// TIA Portal V17 export
// export: Created 2025-03-07T09:17:15.516667Z, ExportSetting WithDefaults, DisplayName Totally Integrated Automation Portal, DisplayVersion V17 Update 8, DisplayName TIA Portal Openness, DisplayVersion V17 Update 8, DisplayName TIA Portal Version Control Interface, DisplayVersion V17, DisplayName SINAMICS Startdrive Advanced, DisplayVersion V17 SP2, DisplayName SINAMICS Startdrive G110M, G120, G120C, G120D, G120P, G115D, DisplayVersion V17 SP2, DisplayName SINAMICS Startdrive G130, G150, S120, S150, SINAMICS MV, S210, DisplayVersion V17 SP2, DisplayName STEP 7 Professional, DisplayVersion V17 Update 8, DisplayName SINUMERIK ONE STEP 7 Toolbox, DisplayVersion V17 Update 12, DisplayName SINUMERIK 840D sl STEP 7 Toolbox, DisplayVersion V17 Update 12, DisplayName STEP 7 Safety, DisplayVersion V17 Update 6, DisplayName WinCC Advanced, DisplayVersion V17 Update 8
FUNCTION "FC355_NCK_M_CH3_UNIT_1_STA_4" : Void   // FC355, LAD
TITLE = Channel 1 data
{ S7_Optimized_Access := 'FALSE' }
AUTHOR : ETXETAR
VERSION : 1.0
// stored: AutoNumber false, IsIECCheckEnabled false, SetENOAutomatically false, UDAEnableTagReadback false
BEGIN

REGION Network 1: ACKNOWLEDGE M700-FIXTURE 4 CLAMP SEQUENCE (READ-IN DISABLE) / ACKNOWLEDGE M100-CLAMP SEQUENCE FIXTURE 1
   // NOTE: WHEN THERE IS NOT INDEXING TABLE AVAILABLE IN THE MACHINE DELETE 
   // DB2171.DBX5.0 AND DB2171.DBX2.0
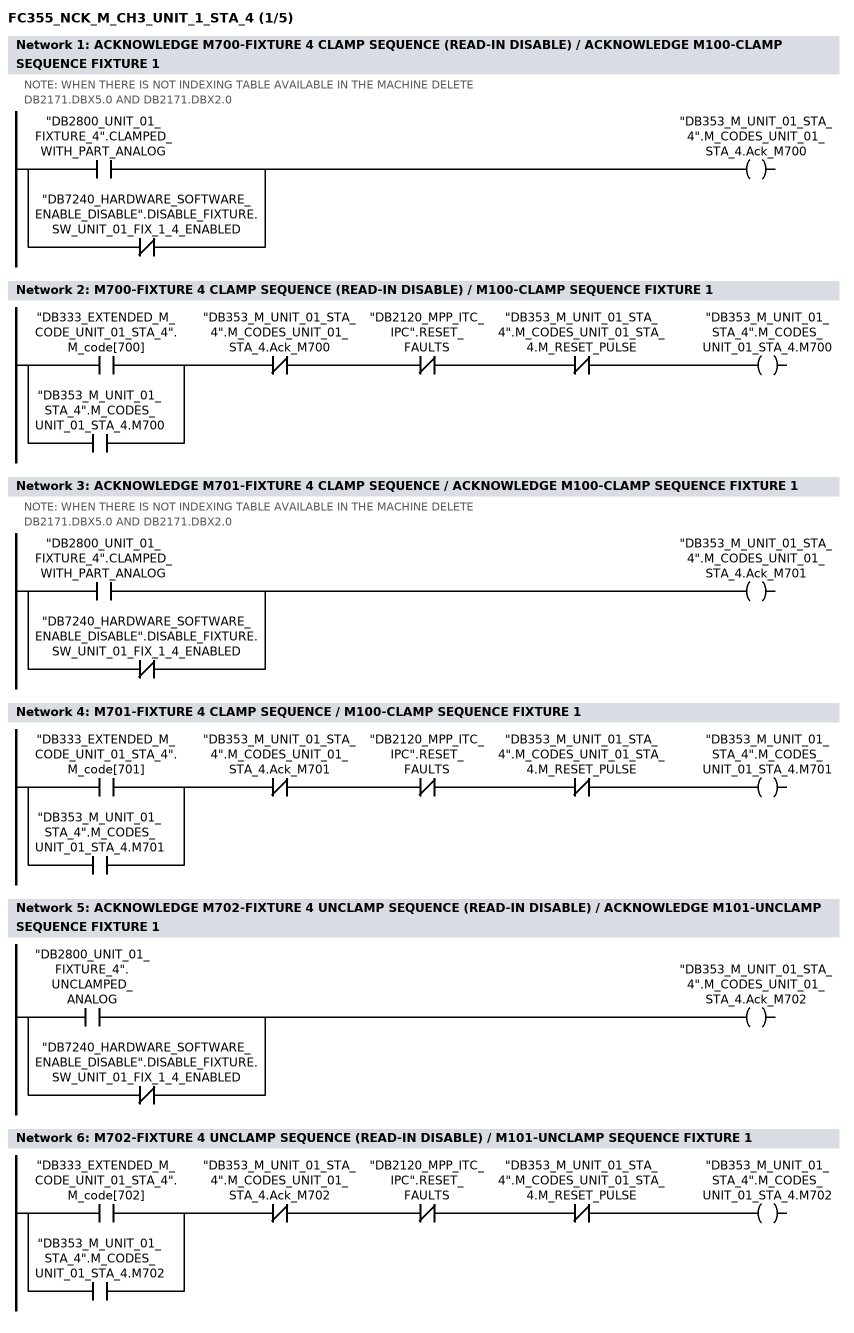
   RUNG wire#powerrail
      Contact( "DB2800_UNIT_01_FIXTURE_4".CLAMPED_WITH_PART_ANALOG )
      wire#w1
      Coil( "DB353_M_UNIT_01_STA_4".M_CODES_UNIT_01_STA_4.Ack_M700 )
   END_RUNG
   RUNG wire#powerrail
      I_Contact( "DB7240_HARDWARE_SOFTWARE_ENABLE_DISABLE".DISABLE_FIXTURE.SW_UNIT_01_FIX_1_4_ENABLED )
   END_RUNG wire#w1
   // the same network as SCL:
   "DB353_M_UNIT_01_STA_4".M_CODES_UNIT_01_STA_4.Ack_M700 := "DB2800_UNIT_01_FIXTURE_4".CLAMPED_WITH_PART_ANALOG OR NOT "DB7240_HARDWARE_SOFTWARE_ENABLE_DISABLE".DISABLE_FIXTURE.SW_UNIT_01_FIX_1_4_ENABLED;
END_REGION

REGION Network 2: M700-FIXTURE 4 CLAMP SEQUENCE (READ-IN DISABLE) / M100-CLAMP SEQUENCE FIXTURE 1
   RUNG wire#powerrail
      Contact( "DB333_EXTENDED_M_CODE_UNIT_01_STA_4".M_code[700] )
      wire#w1
      I_Contact( "DB353_M_UNIT_01_STA_4".M_CODES_UNIT_01_STA_4.Ack_M700 )
      I_Contact( "DB2120_MPP_ITC_IPC".RESET_FAULTS )
      I_Contact( "DB353_M_UNIT_01_STA_4".M_CODES_UNIT_01_STA_4.M_RESET_PULSE )
      Coil( "DB353_M_UNIT_01_STA_4".M_CODES_UNIT_01_STA_4.M700 )
   END_RUNG
   RUNG wire#powerrail
      Contact( "DB353_M_UNIT_01_STA_4".M_CODES_UNIT_01_STA_4.M700 )
   END_RUNG wire#w1
   // the same network as SCL:
   "DB353_M_UNIT_01_STA_4".M_CODES_UNIT_01_STA_4.M700 := ("DB333_EXTENDED_M_CODE_UNIT_01_STA_4".M_code[700] OR "DB353_M_UNIT_01_STA_4".M_CODES_UNIT_01_STA_4.M700) AND NOT "DB353_M_UNIT_01_STA_4".M_CODES_UNIT_01_STA_4.Ack_M700 AND NOT "DB2120_MPP_ITC_IPC".RESET_FAULTS AND NOT "DB353_M_UNIT_01_STA_4".M_CODES_UNIT_01_STA_4.M_RESET_PULSE;
END_REGION

REGION Network 3: ACKNOWLEDGE M701-FIXTURE 4 CLAMP SEQUENCE / ACKNOWLEDGE M100-CLAMP SEQUENCE FIXTURE 1
   // NOTE: WHEN THERE IS NOT INDEXING TABLE AVAILABLE IN THE MACHINE DELETE 
   // DB2171.DBX5.0 AND DB2171.DBX2.0
   RUNG wire#powerrail
      Contact( "DB2800_UNIT_01_FIXTURE_4".CLAMPED_WITH_PART_ANALOG )
      wire#w1
      Coil( "DB353_M_UNIT_01_STA_4".M_CODES_UNIT_01_STA_4.Ack_M701 )
   END_RUNG
   RUNG wire#powerrail
      I_Contact( "DB7240_HARDWARE_SOFTWARE_ENABLE_DISABLE".DISABLE_FIXTURE.SW_UNIT_01_FIX_1_4_ENABLED )
   END_RUNG wire#w1
   // the same network as SCL:
   "DB353_M_UNIT_01_STA_4".M_CODES_UNIT_01_STA_4.Ack_M701 := "DB2800_UNIT_01_FIXTURE_4".CLAMPED_WITH_PART_ANALOG OR NOT "DB7240_HARDWARE_SOFTWARE_ENABLE_DISABLE".DISABLE_FIXTURE.SW_UNIT_01_FIX_1_4_ENABLED;
END_REGION

REGION Network 4: M701-FIXTURE 4 CLAMP SEQUENCE / M100-CLAMP SEQUENCE FIXTURE 1
   RUNG wire#powerrail
      Contact( "DB333_EXTENDED_M_CODE_UNIT_01_STA_4".M_code[701] )
      wire#w1
      I_Contact( "DB353_M_UNIT_01_STA_4".M_CODES_UNIT_01_STA_4.Ack_M701 )
      I_Contact( "DB2120_MPP_ITC_IPC".RESET_FAULTS )
      I_Contact( "DB353_M_UNIT_01_STA_4".M_CODES_UNIT_01_STA_4.M_RESET_PULSE )
      Coil( "DB353_M_UNIT_01_STA_4".M_CODES_UNIT_01_STA_4.M701 )
   END_RUNG
   RUNG wire#powerrail
      Contact( "DB353_M_UNIT_01_STA_4".M_CODES_UNIT_01_STA_4.M701 )
   END_RUNG wire#w1
   // the same network as SCL:
   "DB353_M_UNIT_01_STA_4".M_CODES_UNIT_01_STA_4.M701 := ("DB333_EXTENDED_M_CODE_UNIT_01_STA_4".M_code[701] OR "DB353_M_UNIT_01_STA_4".M_CODES_UNIT_01_STA_4.M701) AND NOT "DB353_M_UNIT_01_STA_4".M_CODES_UNIT_01_STA_4.Ack_M701 AND NOT "DB2120_MPP_ITC_IPC".RESET_FAULTS AND NOT "DB353_M_UNIT_01_STA_4".M_CODES_UNIT_01_STA_4.M_RESET_PULSE;
END_REGION

REGION Network 5: ACKNOWLEDGE M702-FIXTURE 4 UNCLAMP SEQUENCE (READ-IN DISABLE) / ACKNOWLEDGE M101-UNCLAMP SEQUENCE FIXTURE 1
   RUNG wire#powerrail
      Contact( "DB2800_UNIT_01_FIXTURE_4".UNCLAMPED_ANALOG )
      wire#w1
      Coil( "DB353_M_UNIT_01_STA_4".M_CODES_UNIT_01_STA_4.Ack_M702 )
   END_RUNG
   RUNG wire#powerrail
      I_Contact( "DB7240_HARDWARE_SOFTWARE_ENABLE_DISABLE".DISABLE_FIXTURE.SW_UNIT_01_FIX_1_4_ENABLED )
   END_RUNG wire#w1
   // the same network as SCL:
   "DB353_M_UNIT_01_STA_4".M_CODES_UNIT_01_STA_4.Ack_M702 := "DB2800_UNIT_01_FIXTURE_4".UNCLAMPED_ANALOG OR NOT "DB7240_HARDWARE_SOFTWARE_ENABLE_DISABLE".DISABLE_FIXTURE.SW_UNIT_01_FIX_1_4_ENABLED;
END_REGION

REGION Network 6: M702-FIXTURE 4 UNCLAMP SEQUENCE (READ-IN DISABLE) / M101-UNCLAMP SEQUENCE FIXTURE 1
   RUNG wire#powerrail
      Contact( "DB333_EXTENDED_M_CODE_UNIT_01_STA_4".M_code[702] )
      wire#w1
      I_Contact( "DB353_M_UNIT_01_STA_4".M_CODES_UNIT_01_STA_4.Ack_M702 )
      I_Contact( "DB2120_MPP_ITC_IPC".RESET_FAULTS )
      I_Contact( "DB353_M_UNIT_01_STA_4".M_CODES_UNIT_01_STA_4.M_RESET_PULSE )
      Coil( "DB353_M_UNIT_01_STA_4".M_CODES_UNIT_01_STA_4.M702 )
   END_RUNG
   RUNG wire#powerrail
      Contact( "DB353_M_UNIT_01_STA_4".M_CODES_UNIT_01_STA_4.M702 )
   END_RUNG wire#w1
   // the same network as SCL:
   "DB353_M_UNIT_01_STA_4".M_CODES_UNIT_01_STA_4.M702 := ("DB333_EXTENDED_M_CODE_UNIT_01_STA_4".M_code[702] OR "DB353_M_UNIT_01_STA_4".M_CODES_UNIT_01_STA_4.M702) AND NOT "DB353_M_UNIT_01_STA_4".M_CODES_UNIT_01_STA_4.Ack_M702 AND NOT "DB2120_MPP_ITC_IPC".RESET_FAULTS AND NOT "DB353_M_UNIT_01_STA_4".M_CODES_UNIT_01_STA_4.M_RESET_PULSE;
END_REGION

REGION Network 7: ACKNOWLEDGE M703-FIXTURE 4 UNCLAMP SEQUENCE / ACKNOWLEDGE M101-UNCLAMP SEQUENCE FIXTURE 1
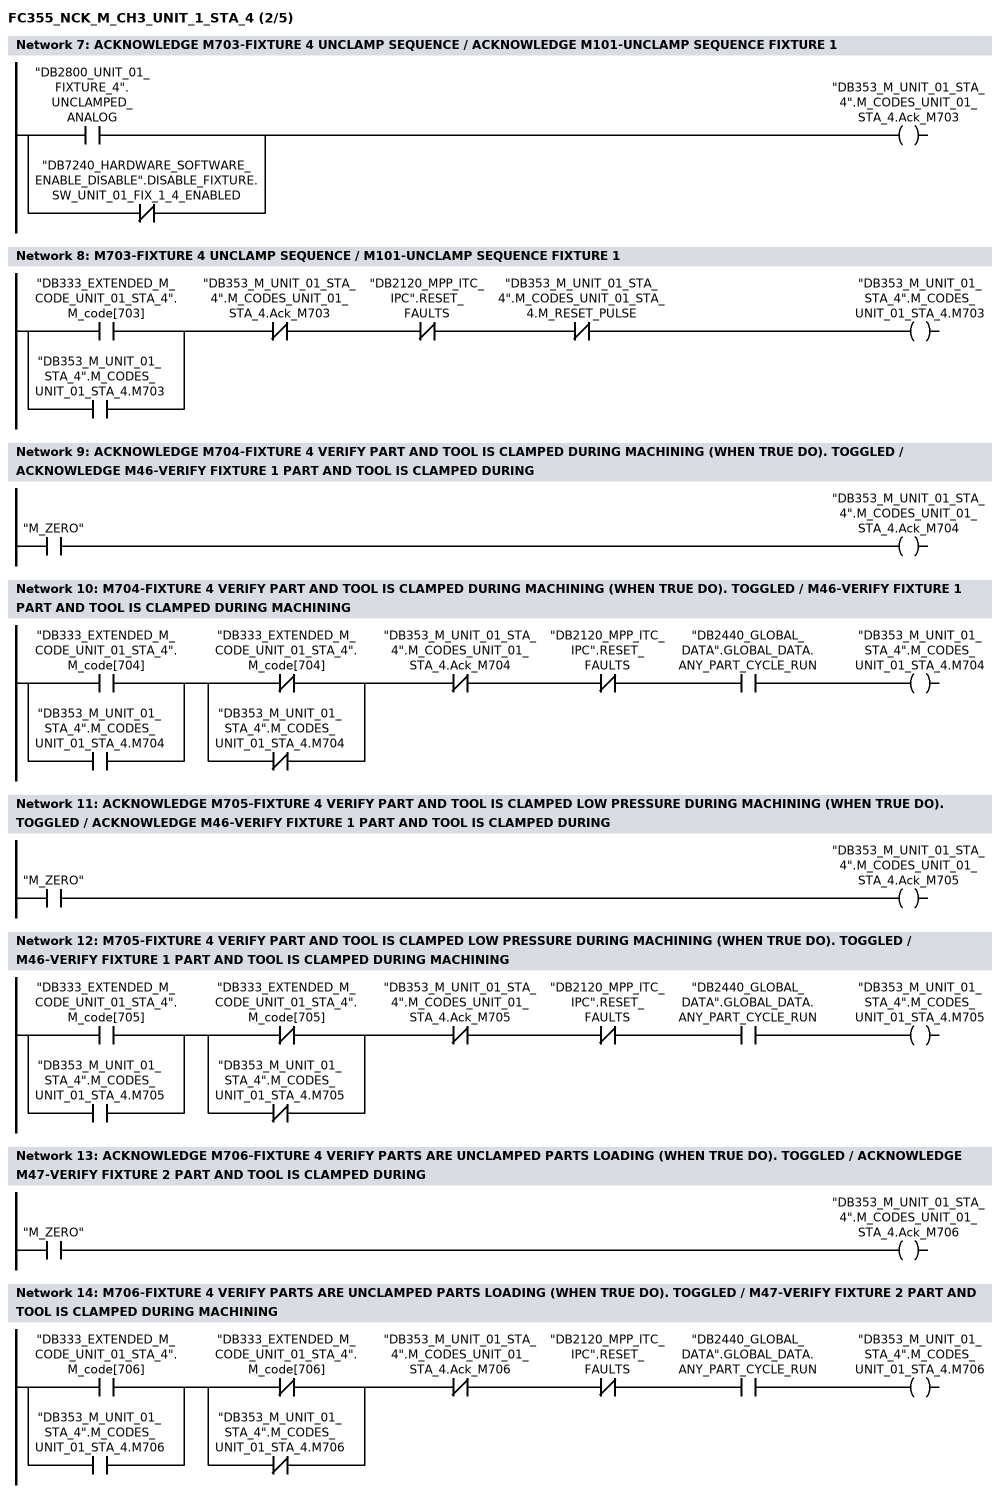
   RUNG wire#powerrail
      Contact( "DB2800_UNIT_01_FIXTURE_4".UNCLAMPED_ANALOG )
      wire#w1
      Coil( "DB353_M_UNIT_01_STA_4".M_CODES_UNIT_01_STA_4.Ack_M703 )
   END_RUNG
   RUNG wire#powerrail
      I_Contact( "DB7240_HARDWARE_SOFTWARE_ENABLE_DISABLE".DISABLE_FIXTURE.SW_UNIT_01_FIX_1_4_ENABLED )
   END_RUNG wire#w1
   // the same network as SCL:
   "DB353_M_UNIT_01_STA_4".M_CODES_UNIT_01_STA_4.Ack_M703 := "DB2800_UNIT_01_FIXTURE_4".UNCLAMPED_ANALOG OR NOT "DB7240_HARDWARE_SOFTWARE_ENABLE_DISABLE".DISABLE_FIXTURE.SW_UNIT_01_FIX_1_4_ENABLED;
END_REGION

REGION Network 8: M703-FIXTURE 4 UNCLAMP SEQUENCE / M101-UNCLAMP SEQUENCE FIXTURE 1
   RUNG wire#powerrail
      Contact( "DB333_EXTENDED_M_CODE_UNIT_01_STA_4".M_code[703] )
      wire#w1
      I_Contact( "DB353_M_UNIT_01_STA_4".M_CODES_UNIT_01_STA_4.Ack_M703 )
      I_Contact( "DB2120_MPP_ITC_IPC".RESET_FAULTS )
      I_Contact( "DB353_M_UNIT_01_STA_4".M_CODES_UNIT_01_STA_4.M_RESET_PULSE )
      Coil( "DB353_M_UNIT_01_STA_4".M_CODES_UNIT_01_STA_4.M703 )
   END_RUNG
   RUNG wire#powerrail
      Contact( "DB353_M_UNIT_01_STA_4".M_CODES_UNIT_01_STA_4.M703 )
   END_RUNG wire#w1
   // the same network as SCL:
   "DB353_M_UNIT_01_STA_4".M_CODES_UNIT_01_STA_4.M703 := ("DB333_EXTENDED_M_CODE_UNIT_01_STA_4".M_code[703] OR "DB353_M_UNIT_01_STA_4".M_CODES_UNIT_01_STA_4.M703) AND NOT "DB353_M_UNIT_01_STA_4".M_CODES_UNIT_01_STA_4.Ack_M703 AND NOT "DB2120_MPP_ITC_IPC".RESET_FAULTS AND NOT "DB353_M_UNIT_01_STA_4".M_CODES_UNIT_01_STA_4.M_RESET_PULSE;
END_REGION

REGION Network 9: ACKNOWLEDGE M704-FIXTURE 4 VERIFY PART AND TOOL IS CLAMPED DURING MACHINING (WHEN TRUE DO). TOGGLED / ACKNOWLEDGE M46-VERIFY FIXTURE 1 PART AND TOOL IS CLAMPED DURING
   RUNG wire#powerrail
      Contact( "M_ZERO" )
      Coil( "DB353_M_UNIT_01_STA_4".M_CODES_UNIT_01_STA_4.Ack_M704 )
   END_RUNG
   // the same network as SCL:
   "DB353_M_UNIT_01_STA_4".M_CODES_UNIT_01_STA_4.Ack_M704 := "M_ZERO";
END_REGION

REGION Network 10: M704-FIXTURE 4 VERIFY PART AND TOOL IS CLAMPED DURING MACHINING (WHEN TRUE DO). TOGGLED / M46-VERIFY FIXTURE 1 PART AND TOOL IS CLAMPED DURING MACHINING
   RUNG wire#powerrail
      Contact( "DB333_EXTENDED_M_CODE_UNIT_01_STA_4".M_code[704] )
      wire#w1
      I_Contact( "DB333_EXTENDED_M_CODE_UNIT_01_STA_4".M_code[704] )
      wire#w2
      I_Contact( "DB353_M_UNIT_01_STA_4".M_CODES_UNIT_01_STA_4.Ack_M704 )
      I_Contact( "DB2120_MPP_ITC_IPC".RESET_FAULTS )
      Contact( "DB2440_GLOBAL_DATA".GLOBAL_DATA.ANY_PART_CYCLE_RUN )
      Coil( "DB353_M_UNIT_01_STA_4".M_CODES_UNIT_01_STA_4.M704 )
   END_RUNG
   RUNG wire#powerrail
      Contact( "DB353_M_UNIT_01_STA_4".M_CODES_UNIT_01_STA_4.M704 )
   END_RUNG wire#w1
   RUNG wire#w1
      I_Contact( "DB353_M_UNIT_01_STA_4".M_CODES_UNIT_01_STA_4.M704 )
   END_RUNG wire#w2
   // the same network as SCL:
   "DB353_M_UNIT_01_STA_4".M_CODES_UNIT_01_STA_4.M704 := ("DB333_EXTENDED_M_CODE_UNIT_01_STA_4".M_code[704] OR "DB353_M_UNIT_01_STA_4".M_CODES_UNIT_01_STA_4.M704) AND (NOT "DB333_EXTENDED_M_CODE_UNIT_01_STA_4".M_code[704] OR NOT "DB353_M_UNIT_01_STA_4".M_CODES_UNIT_01_STA_4.M704) AND NOT "DB353_M_UNIT_01_STA_4".M_CODES_UNIT_01_STA_4.Ack_M704 AND NOT "DB2120_MPP_ITC_IPC".RESET_FAULTS AND "DB2440_GLOBAL_DATA".GLOBAL_DATA.ANY_PART_CYCLE_RUN;
END_REGION

REGION Network 11: ACKNOWLEDGE M705-FIXTURE 4 VERIFY PART AND TOOL IS CLAMPED LOW PRESSURE DURING MACHINING (WHEN TRUE DO). TOGGLED / ACKNOWLEDGE M46-VERIFY FIXTURE 1 PART AND TOOL IS CLAMPED DURING
   RUNG wire#powerrail
      Contact( "M_ZERO" )
      Coil( "DB353_M_UNIT_01_STA_4".M_CODES_UNIT_01_STA_4.Ack_M705 )
   END_RUNG
   // the same network as SCL:
   "DB353_M_UNIT_01_STA_4".M_CODES_UNIT_01_STA_4.Ack_M705 := "M_ZERO";
END_REGION

REGION Network 12: M705-FIXTURE 4 VERIFY PART AND TOOL IS CLAMPED LOW PRESSURE DURING MACHINING (WHEN TRUE DO). TOGGLED / M46-VERIFY FIXTURE 1 PART AND TOOL IS CLAMPED DURING MACHINING
   RUNG wire#powerrail
      Contact( "DB333_EXTENDED_M_CODE_UNIT_01_STA_4".M_code[705] )
      wire#w1
      I_Contact( "DB333_EXTENDED_M_CODE_UNIT_01_STA_4".M_code[705] )
      wire#w2
      I_Contact( "DB353_M_UNIT_01_STA_4".M_CODES_UNIT_01_STA_4.Ack_M705 )
      I_Contact( "DB2120_MPP_ITC_IPC".RESET_FAULTS )
      Contact( "DB2440_GLOBAL_DATA".GLOBAL_DATA.ANY_PART_CYCLE_RUN )
      Coil( "DB353_M_UNIT_01_STA_4".M_CODES_UNIT_01_STA_4.M705 )
   END_RUNG
   RUNG wire#powerrail
      Contact( "DB353_M_UNIT_01_STA_4".M_CODES_UNIT_01_STA_4.M705 )
   END_RUNG wire#w1
   RUNG wire#w1
      I_Contact( "DB353_M_UNIT_01_STA_4".M_CODES_UNIT_01_STA_4.M705 )
   END_RUNG wire#w2
   // the same network as SCL:
   "DB353_M_UNIT_01_STA_4".M_CODES_UNIT_01_STA_4.M705 := ("DB333_EXTENDED_M_CODE_UNIT_01_STA_4".M_code[705] OR "DB353_M_UNIT_01_STA_4".M_CODES_UNIT_01_STA_4.M705) AND (NOT "DB333_EXTENDED_M_CODE_UNIT_01_STA_4".M_code[705] OR NOT "DB353_M_UNIT_01_STA_4".M_CODES_UNIT_01_STA_4.M705) AND NOT "DB353_M_UNIT_01_STA_4".M_CODES_UNIT_01_STA_4.Ack_M705 AND NOT "DB2120_MPP_ITC_IPC".RESET_FAULTS AND "DB2440_GLOBAL_DATA".GLOBAL_DATA.ANY_PART_CYCLE_RUN;
END_REGION

REGION Network 13: ACKNOWLEDGE M706-FIXTURE 4 VERIFY PARTS ARE UNCLAMPED PARTS LOADING (WHEN TRUE DO). TOGGLED / ACKNOWLEDGE M47-VERIFY FIXTURE 2 PART AND TOOL IS CLAMPED DURING
   RUNG wire#powerrail
      Contact( "M_ZERO" )
      Coil( "DB353_M_UNIT_01_STA_4".M_CODES_UNIT_01_STA_4.Ack_M706 )
   END_RUNG
   // the same network as SCL:
   "DB353_M_UNIT_01_STA_4".M_CODES_UNIT_01_STA_4.Ack_M706 := "M_ZERO";
END_REGION

REGION Network 14: M706-FIXTURE 4 VERIFY PARTS ARE UNCLAMPED PARTS LOADING (WHEN TRUE DO). TOGGLED / M47-VERIFY FIXTURE 2 PART AND TOOL IS CLAMPED DURING MACHINING
   RUNG wire#powerrail
      Contact( "DB333_EXTENDED_M_CODE_UNIT_01_STA_4".M_code[706] )
      wire#w1
      I_Contact( "DB333_EXTENDED_M_CODE_UNIT_01_STA_4".M_code[706] )
      wire#w2
      I_Contact( "DB353_M_UNIT_01_STA_4".M_CODES_UNIT_01_STA_4.Ack_M706 )
      I_Contact( "DB2120_MPP_ITC_IPC".RESET_FAULTS )
      Contact( "DB2440_GLOBAL_DATA".GLOBAL_DATA.ANY_PART_CYCLE_RUN )
      Coil( "DB353_M_UNIT_01_STA_4".M_CODES_UNIT_01_STA_4.M706 )
   END_RUNG
   RUNG wire#powerrail
      Contact( "DB353_M_UNIT_01_STA_4".M_CODES_UNIT_01_STA_4.M706 )
   END_RUNG wire#w1
   RUNG wire#w1
      I_Contact( "DB353_M_UNIT_01_STA_4".M_CODES_UNIT_01_STA_4.M706 )
   END_RUNG wire#w2
   // the same network as SCL:
   "DB353_M_UNIT_01_STA_4".M_CODES_UNIT_01_STA_4.M706 := ("DB333_EXTENDED_M_CODE_UNIT_01_STA_4".M_code[706] OR "DB353_M_UNIT_01_STA_4".M_CODES_UNIT_01_STA_4.M706) AND (NOT "DB333_EXTENDED_M_CODE_UNIT_01_STA_4".M_code[706] OR NOT "DB353_M_UNIT_01_STA_4".M_CODES_UNIT_01_STA_4.M706) AND NOT "DB353_M_UNIT_01_STA_4".M_CODES_UNIT_01_STA_4.Ack_M706 AND NOT "DB2120_MPP_ITC_IPC".RESET_FAULTS AND "DB2440_GLOBAL_DATA".GLOBAL_DATA.ANY_PART_CYCLE_RUN;
END_REGION

REGION Network 15: ACKNOWLEDGE M707-FIXTURE 4 VERIFY FIXTURE REMAINS CLAMPED
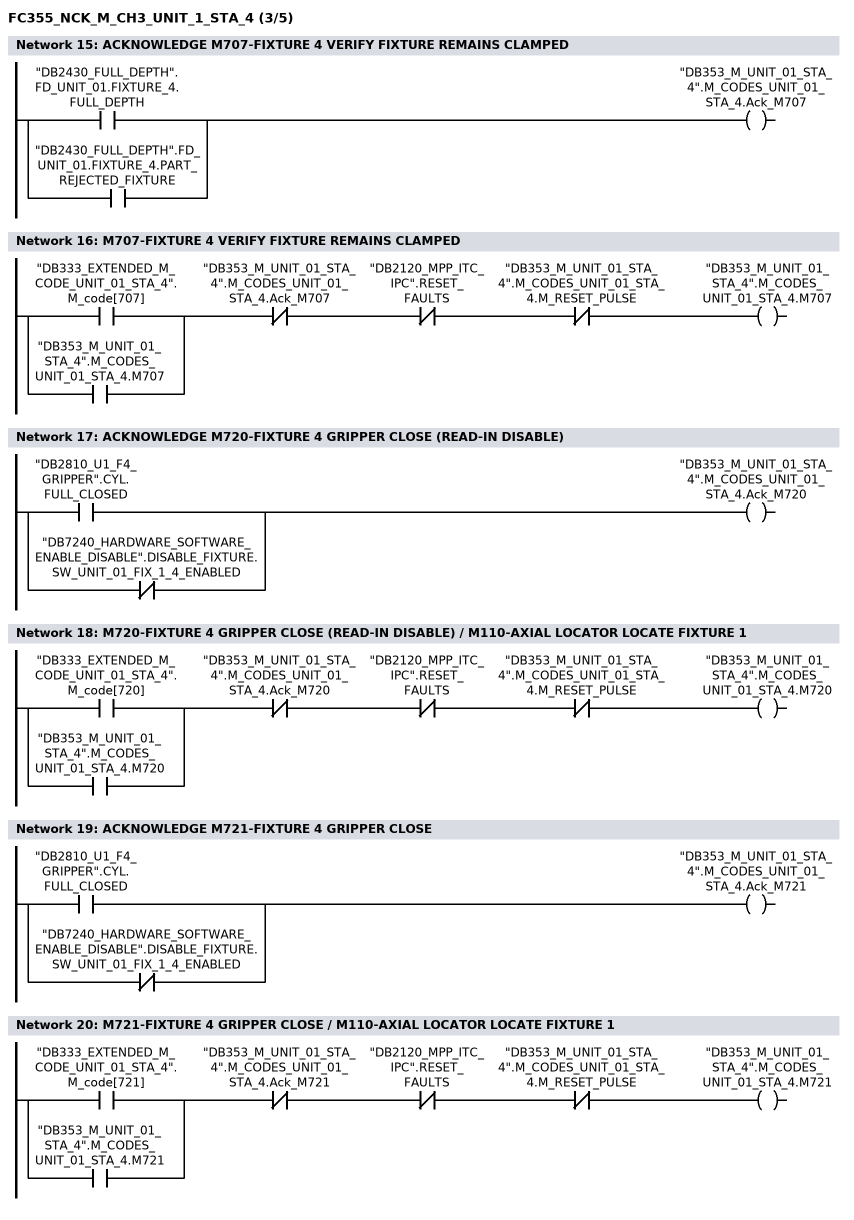
   RUNG wire#powerrail
      Contact( "DB2430_FULL_DEPTH".FD_UNIT_01.FIXTURE_4.FULL_DEPTH )
      wire#w1
      Coil( "DB353_M_UNIT_01_STA_4".M_CODES_UNIT_01_STA_4.Ack_M707 )
   END_RUNG
   RUNG wire#powerrail
      Contact( "DB2430_FULL_DEPTH".FD_UNIT_01.FIXTURE_4.PART_REJECTED_FIXTURE )
   END_RUNG wire#w1
   // the same network as SCL:
   "DB353_M_UNIT_01_STA_4".M_CODES_UNIT_01_STA_4.Ack_M707 := "DB2430_FULL_DEPTH".FD_UNIT_01.FIXTURE_4.FULL_DEPTH OR "DB2430_FULL_DEPTH".FD_UNIT_01.FIXTURE_4.PART_REJECTED_FIXTURE;
END_REGION

REGION Network 16: M707-FIXTURE 4 VERIFY FIXTURE REMAINS CLAMPED
   RUNG wire#powerrail
      Contact( "DB333_EXTENDED_M_CODE_UNIT_01_STA_4".M_code[707] )
      wire#w1
      I_Contact( "DB353_M_UNIT_01_STA_4".M_CODES_UNIT_01_STA_4.Ack_M707 )
      I_Contact( "DB2120_MPP_ITC_IPC".RESET_FAULTS )
      I_Contact( "DB353_M_UNIT_01_STA_4".M_CODES_UNIT_01_STA_4.M_RESET_PULSE )
      Coil( "DB353_M_UNIT_01_STA_4".M_CODES_UNIT_01_STA_4.M707 )
   END_RUNG
   RUNG wire#powerrail
      Contact( "DB353_M_UNIT_01_STA_4".M_CODES_UNIT_01_STA_4.M707 )
   END_RUNG wire#w1
   // the same network as SCL:
   "DB353_M_UNIT_01_STA_4".M_CODES_UNIT_01_STA_4.M707 := ("DB333_EXTENDED_M_CODE_UNIT_01_STA_4".M_code[707] OR "DB353_M_UNIT_01_STA_4".M_CODES_UNIT_01_STA_4.M707) AND NOT "DB353_M_UNIT_01_STA_4".M_CODES_UNIT_01_STA_4.Ack_M707 AND NOT "DB2120_MPP_ITC_IPC".RESET_FAULTS AND NOT "DB353_M_UNIT_01_STA_4".M_CODES_UNIT_01_STA_4.M_RESET_PULSE;
END_REGION

REGION Network 17: ACKNOWLEDGE M720-FIXTURE 4 GRIPPER CLOSE (READ-IN DISABLE)
   RUNG wire#powerrail
      Contact( "DB2810_U1_F4_GRIPPER".CYL.FULL_CLOSED )
      wire#w1
      Coil( "DB353_M_UNIT_01_STA_4".M_CODES_UNIT_01_STA_4.Ack_M720 )
   END_RUNG
   RUNG wire#powerrail
      I_Contact( "DB7240_HARDWARE_SOFTWARE_ENABLE_DISABLE".DISABLE_FIXTURE.SW_UNIT_01_FIX_1_4_ENABLED )
   END_RUNG wire#w1
   // the same network as SCL:
   "DB353_M_UNIT_01_STA_4".M_CODES_UNIT_01_STA_4.Ack_M720 := "DB2810_U1_F4_GRIPPER".CYL.FULL_CLOSED OR NOT "DB7240_HARDWARE_SOFTWARE_ENABLE_DISABLE".DISABLE_FIXTURE.SW_UNIT_01_FIX_1_4_ENABLED;
END_REGION

REGION Network 18: M720-FIXTURE 4 GRIPPER CLOSE (READ-IN DISABLE) / M110-AXIAL LOCATOR LOCATE FIXTURE 1
   RUNG wire#powerrail
      Contact( "DB333_EXTENDED_M_CODE_UNIT_01_STA_4".M_code[720] )
      wire#w1
      I_Contact( "DB353_M_UNIT_01_STA_4".M_CODES_UNIT_01_STA_4.Ack_M720 )
      I_Contact( "DB2120_MPP_ITC_IPC".RESET_FAULTS )
      I_Contact( "DB353_M_UNIT_01_STA_4".M_CODES_UNIT_01_STA_4.M_RESET_PULSE )
      Coil( "DB353_M_UNIT_01_STA_4".M_CODES_UNIT_01_STA_4.M720 )
   END_RUNG
   RUNG wire#powerrail
      Contact( "DB353_M_UNIT_01_STA_4".M_CODES_UNIT_01_STA_4.M720 )
   END_RUNG wire#w1
   // the same network as SCL:
   "DB353_M_UNIT_01_STA_4".M_CODES_UNIT_01_STA_4.M720 := ("DB333_EXTENDED_M_CODE_UNIT_01_STA_4".M_code[720] OR "DB353_M_UNIT_01_STA_4".M_CODES_UNIT_01_STA_4.M720) AND NOT "DB353_M_UNIT_01_STA_4".M_CODES_UNIT_01_STA_4.Ack_M720 AND NOT "DB2120_MPP_ITC_IPC".RESET_FAULTS AND NOT "DB353_M_UNIT_01_STA_4".M_CODES_UNIT_01_STA_4.M_RESET_PULSE;
END_REGION

REGION Network 19: ACKNOWLEDGE M721-FIXTURE 4 GRIPPER CLOSE
   RUNG wire#powerrail
      Contact( "DB2810_U1_F4_GRIPPER".CYL.FULL_CLOSED )
      wire#w1
      Coil( "DB353_M_UNIT_01_STA_4".M_CODES_UNIT_01_STA_4.Ack_M721 )
   END_RUNG
   RUNG wire#powerrail
      I_Contact( "DB7240_HARDWARE_SOFTWARE_ENABLE_DISABLE".DISABLE_FIXTURE.SW_UNIT_01_FIX_1_4_ENABLED )
   END_RUNG wire#w1
   // the same network as SCL:
   "DB353_M_UNIT_01_STA_4".M_CODES_UNIT_01_STA_4.Ack_M721 := "DB2810_U1_F4_GRIPPER".CYL.FULL_CLOSED OR NOT "DB7240_HARDWARE_SOFTWARE_ENABLE_DISABLE".DISABLE_FIXTURE.SW_UNIT_01_FIX_1_4_ENABLED;
END_REGION

REGION Network 20: M721-FIXTURE 4 GRIPPER CLOSE / M110-AXIAL LOCATOR LOCATE FIXTURE 1
   RUNG wire#powerrail
      Contact( "DB333_EXTENDED_M_CODE_UNIT_01_STA_4".M_code[721] )
      wire#w1
      I_Contact( "DB353_M_UNIT_01_STA_4".M_CODES_UNIT_01_STA_4.Ack_M721 )
      I_Contact( "DB2120_MPP_ITC_IPC".RESET_FAULTS )
      I_Contact( "DB353_M_UNIT_01_STA_4".M_CODES_UNIT_01_STA_4.M_RESET_PULSE )
      Coil( "DB353_M_UNIT_01_STA_4".M_CODES_UNIT_01_STA_4.M721 )
   END_RUNG
   RUNG wire#powerrail
      Contact( "DB353_M_UNIT_01_STA_4".M_CODES_UNIT_01_STA_4.M721 )
   END_RUNG wire#w1
   // the same network as SCL:
   "DB353_M_UNIT_01_STA_4".M_CODES_UNIT_01_STA_4.M721 := ("DB333_EXTENDED_M_CODE_UNIT_01_STA_4".M_code[721] OR "DB353_M_UNIT_01_STA_4".M_CODES_UNIT_01_STA_4.M721) AND NOT "DB353_M_UNIT_01_STA_4".M_CODES_UNIT_01_STA_4.Ack_M721 AND NOT "DB2120_MPP_ITC_IPC".RESET_FAULTS AND NOT "DB353_M_UNIT_01_STA_4".M_CODES_UNIT_01_STA_4.M_RESET_PULSE;
END_REGION

REGION Network 21: ACKNOWLEDGE M722-FIXTURE 4 GRIPPER RETURN (READ-IN DISABLE) / ACKNOWLEDGE M111-AXIAL LOCATOR RETURN FIXTURE 1
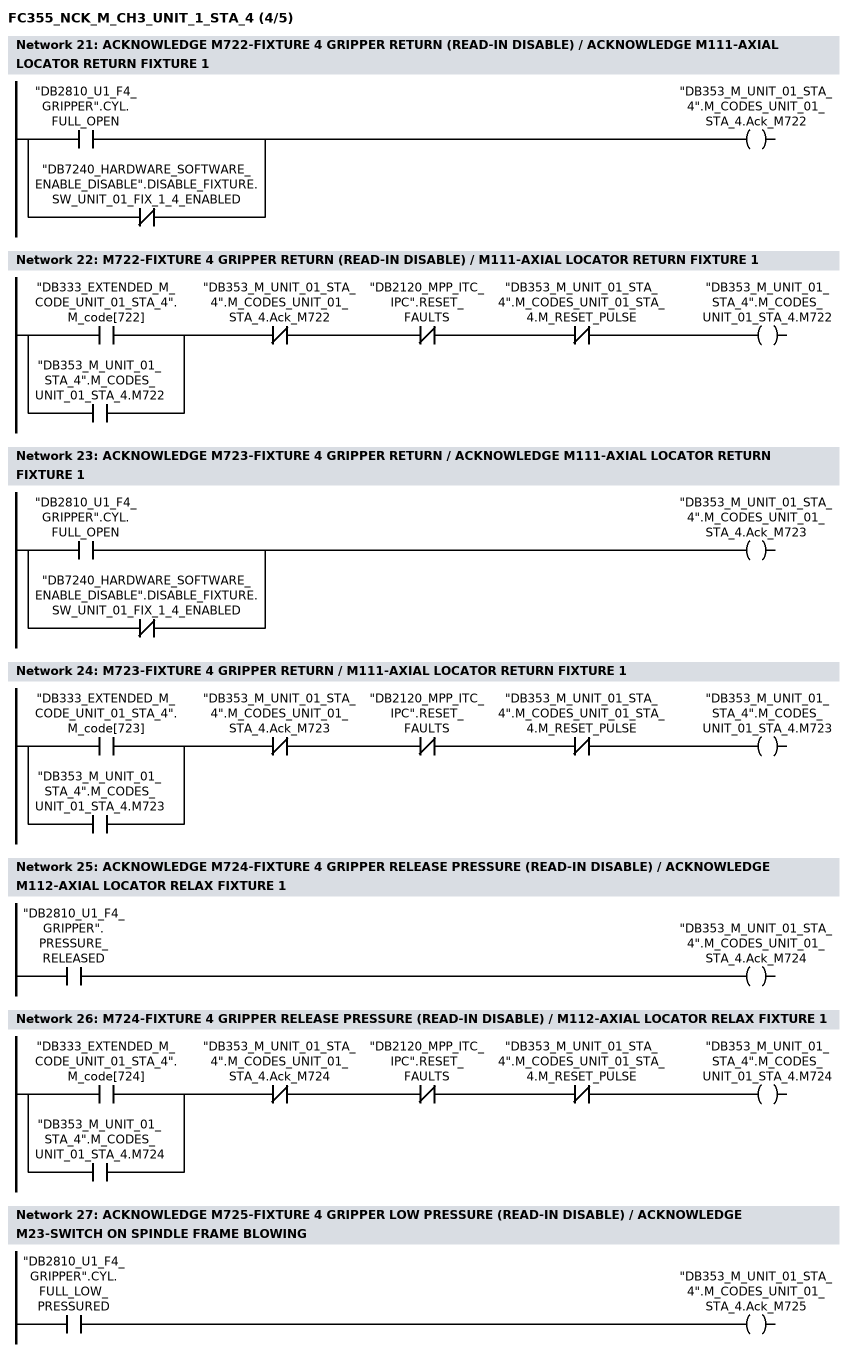
   RUNG wire#powerrail
      Contact( "DB2810_U1_F4_GRIPPER".CYL.FULL_OPEN )
      wire#w1
      Coil( "DB353_M_UNIT_01_STA_4".M_CODES_UNIT_01_STA_4.Ack_M722 )
   END_RUNG
   RUNG wire#powerrail
      I_Contact( "DB7240_HARDWARE_SOFTWARE_ENABLE_DISABLE".DISABLE_FIXTURE.SW_UNIT_01_FIX_1_4_ENABLED )
   END_RUNG wire#w1
   // the same network as SCL:
   "DB353_M_UNIT_01_STA_4".M_CODES_UNIT_01_STA_4.Ack_M722 := "DB2810_U1_F4_GRIPPER".CYL.FULL_OPEN OR NOT "DB7240_HARDWARE_SOFTWARE_ENABLE_DISABLE".DISABLE_FIXTURE.SW_UNIT_01_FIX_1_4_ENABLED;
END_REGION

REGION Network 22: M722-FIXTURE 4 GRIPPER RETURN (READ-IN DISABLE) / M111-AXIAL LOCATOR RETURN FIXTURE 1
   RUNG wire#powerrail
      Contact( "DB333_EXTENDED_M_CODE_UNIT_01_STA_4".M_code[722] )
      wire#w1
      I_Contact( "DB353_M_UNIT_01_STA_4".M_CODES_UNIT_01_STA_4.Ack_M722 )
      I_Contact( "DB2120_MPP_ITC_IPC".RESET_FAULTS )
      I_Contact( "DB353_M_UNIT_01_STA_4".M_CODES_UNIT_01_STA_4.M_RESET_PULSE )
      Coil( "DB353_M_UNIT_01_STA_4".M_CODES_UNIT_01_STA_4.M722 )
   END_RUNG
   RUNG wire#powerrail
      Contact( "DB353_M_UNIT_01_STA_4".M_CODES_UNIT_01_STA_4.M722 )
   END_RUNG wire#w1
   // the same network as SCL:
   "DB353_M_UNIT_01_STA_4".M_CODES_UNIT_01_STA_4.M722 := ("DB333_EXTENDED_M_CODE_UNIT_01_STA_4".M_code[722] OR "DB353_M_UNIT_01_STA_4".M_CODES_UNIT_01_STA_4.M722) AND NOT "DB353_M_UNIT_01_STA_4".M_CODES_UNIT_01_STA_4.Ack_M722 AND NOT "DB2120_MPP_ITC_IPC".RESET_FAULTS AND NOT "DB353_M_UNIT_01_STA_4".M_CODES_UNIT_01_STA_4.M_RESET_PULSE;
END_REGION

REGION Network 23: ACKNOWLEDGE M723-FIXTURE 4 GRIPPER RETURN / ACKNOWLEDGE M111-AXIAL LOCATOR RETURN FIXTURE 1
   RUNG wire#powerrail
      Contact( "DB2810_U1_F4_GRIPPER".CYL.FULL_OPEN )
      wire#w1
      Coil( "DB353_M_UNIT_01_STA_4".M_CODES_UNIT_01_STA_4.Ack_M723 )
   END_RUNG
   RUNG wire#powerrail
      I_Contact( "DB7240_HARDWARE_SOFTWARE_ENABLE_DISABLE".DISABLE_FIXTURE.SW_UNIT_01_FIX_1_4_ENABLED )
   END_RUNG wire#w1
   // the same network as SCL:
   "DB353_M_UNIT_01_STA_4".M_CODES_UNIT_01_STA_4.Ack_M723 := "DB2810_U1_F4_GRIPPER".CYL.FULL_OPEN OR NOT "DB7240_HARDWARE_SOFTWARE_ENABLE_DISABLE".DISABLE_FIXTURE.SW_UNIT_01_FIX_1_4_ENABLED;
END_REGION

REGION Network 24: M723-FIXTURE 4 GRIPPER RETURN / M111-AXIAL LOCATOR RETURN FIXTURE 1
   RUNG wire#powerrail
      Contact( "DB333_EXTENDED_M_CODE_UNIT_01_STA_4".M_code[723] )
      wire#w1
      I_Contact( "DB353_M_UNIT_01_STA_4".M_CODES_UNIT_01_STA_4.Ack_M723 )
      I_Contact( "DB2120_MPP_ITC_IPC".RESET_FAULTS )
      I_Contact( "DB353_M_UNIT_01_STA_4".M_CODES_UNIT_01_STA_4.M_RESET_PULSE )
      Coil( "DB353_M_UNIT_01_STA_4".M_CODES_UNIT_01_STA_4.M723 )
   END_RUNG
   RUNG wire#powerrail
      Contact( "DB353_M_UNIT_01_STA_4".M_CODES_UNIT_01_STA_4.M723 )
   END_RUNG wire#w1
   // the same network as SCL:
   "DB353_M_UNIT_01_STA_4".M_CODES_UNIT_01_STA_4.M723 := ("DB333_EXTENDED_M_CODE_UNIT_01_STA_4".M_code[723] OR "DB353_M_UNIT_01_STA_4".M_CODES_UNIT_01_STA_4.M723) AND NOT "DB353_M_UNIT_01_STA_4".M_CODES_UNIT_01_STA_4.Ack_M723 AND NOT "DB2120_MPP_ITC_IPC".RESET_FAULTS AND NOT "DB353_M_UNIT_01_STA_4".M_CODES_UNIT_01_STA_4.M_RESET_PULSE;
END_REGION

REGION Network 25: ACKNOWLEDGE M724-FIXTURE 4 GRIPPER RELEASE PRESSURE (READ-IN DISABLE) / ACKNOWLEDGE M112-AXIAL LOCATOR RELAX FIXTURE 1
   RUNG wire#powerrail
      Contact( "DB2810_U1_F4_GRIPPER".PRESSURE_RELEASED )
      Coil( "DB353_M_UNIT_01_STA_4".M_CODES_UNIT_01_STA_4.Ack_M724 )
   END_RUNG
   // the same network as SCL:
   "DB353_M_UNIT_01_STA_4".M_CODES_UNIT_01_STA_4.Ack_M724 := "DB2810_U1_F4_GRIPPER".PRESSURE_RELEASED;
END_REGION

REGION Network 26: M724-FIXTURE 4 GRIPPER RELEASE PRESSURE (READ-IN DISABLE) / M112-AXIAL LOCATOR RELAX FIXTURE 1
   RUNG wire#powerrail
      Contact( "DB333_EXTENDED_M_CODE_UNIT_01_STA_4".M_code[724] )
      wire#w1
      I_Contact( "DB353_M_UNIT_01_STA_4".M_CODES_UNIT_01_STA_4.Ack_M724 )
      I_Contact( "DB2120_MPP_ITC_IPC".RESET_FAULTS )
      I_Contact( "DB353_M_UNIT_01_STA_4".M_CODES_UNIT_01_STA_4.M_RESET_PULSE )
      Coil( "DB353_M_UNIT_01_STA_4".M_CODES_UNIT_01_STA_4.M724 )
   END_RUNG
   RUNG wire#powerrail
      Contact( "DB353_M_UNIT_01_STA_4".M_CODES_UNIT_01_STA_4.M724 )
   END_RUNG wire#w1
   // the same network as SCL:
   "DB353_M_UNIT_01_STA_4".M_CODES_UNIT_01_STA_4.M724 := ("DB333_EXTENDED_M_CODE_UNIT_01_STA_4".M_code[724] OR "DB353_M_UNIT_01_STA_4".M_CODES_UNIT_01_STA_4.M724) AND NOT "DB353_M_UNIT_01_STA_4".M_CODES_UNIT_01_STA_4.Ack_M724 AND NOT "DB2120_MPP_ITC_IPC".RESET_FAULTS AND NOT "DB353_M_UNIT_01_STA_4".M_CODES_UNIT_01_STA_4.M_RESET_PULSE;
END_REGION

REGION Network 27: ACKNOWLEDGE M725-FIXTURE 4 GRIPPER LOW PRESSURE (READ-IN DISABLE) / ACKNOWLEDGE M23-SWITCH ON SPINDLE FRAME BLOWING
   RUNG wire#powerrail
      Contact( "DB2810_U1_F4_GRIPPER".CYL.FULL_LOW_PRESSURED )
      Coil( "DB353_M_UNIT_01_STA_4".M_CODES_UNIT_01_STA_4.Ack_M725 )
   END_RUNG
   // the same network as SCL:
   "DB353_M_UNIT_01_STA_4".M_CODES_UNIT_01_STA_4.Ack_M725 := "DB2810_U1_F4_GRIPPER".CYL.FULL_LOW_PRESSURED;
END_REGION

REGION Network 28: M725-FIXTURE 4 GRIPPER LOW PRESSURE (READ-IN DISABLE) / M23-SWITCH ON SPINDLE FRAME BLOWING
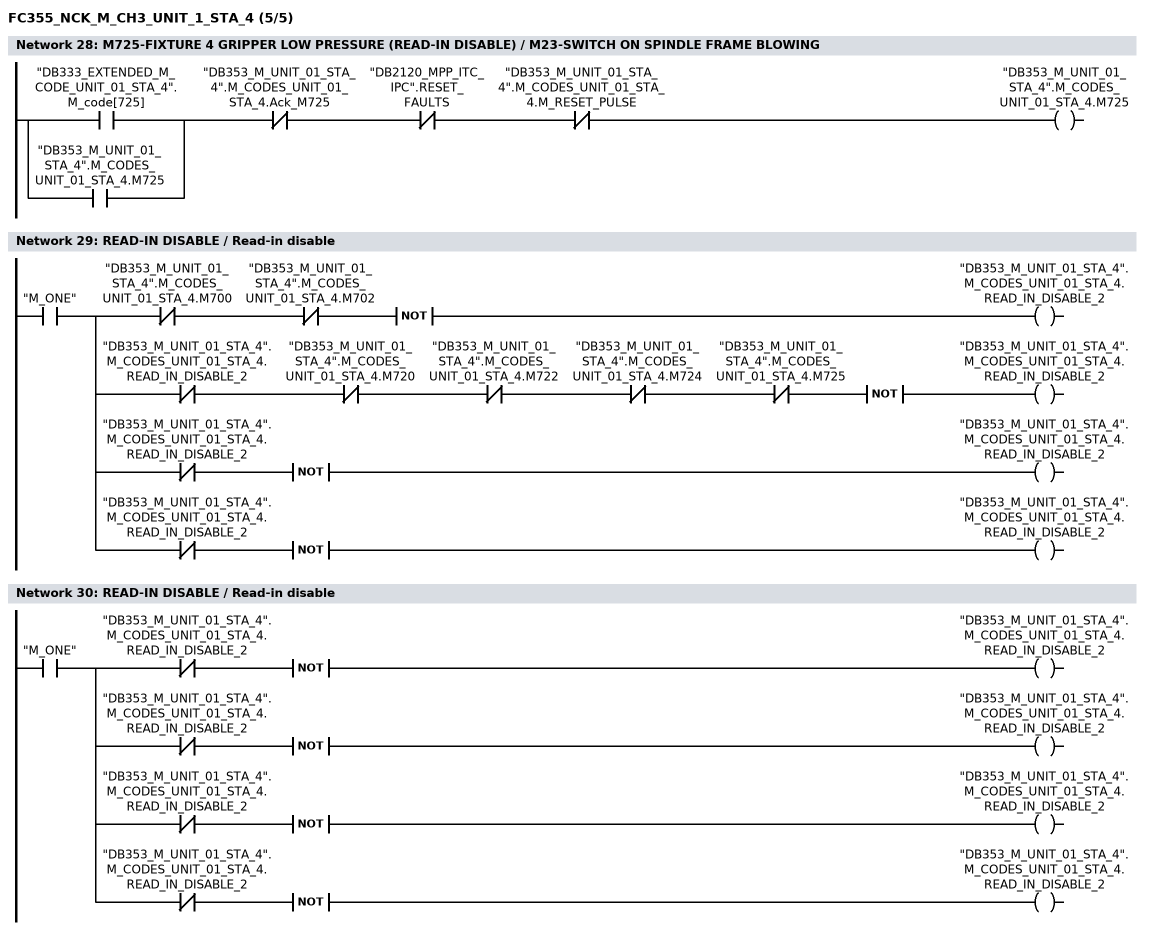
   RUNG wire#powerrail
      Contact( "DB333_EXTENDED_M_CODE_UNIT_01_STA_4".M_code[725] )
      wire#w1
      I_Contact( "DB353_M_UNIT_01_STA_4".M_CODES_UNIT_01_STA_4.Ack_M725 )
      I_Contact( "DB2120_MPP_ITC_IPC".RESET_FAULTS )
      I_Contact( "DB353_M_UNIT_01_STA_4".M_CODES_UNIT_01_STA_4.M_RESET_PULSE )
      Coil( "DB353_M_UNIT_01_STA_4".M_CODES_UNIT_01_STA_4.M725 )
   END_RUNG
   RUNG wire#powerrail
      Contact( "DB353_M_UNIT_01_STA_4".M_CODES_UNIT_01_STA_4.M725 )
   END_RUNG wire#w1
   // the same network as SCL:
   "DB353_M_UNIT_01_STA_4".M_CODES_UNIT_01_STA_4.M725 := ("DB333_EXTENDED_M_CODE_UNIT_01_STA_4".M_code[725] OR "DB353_M_UNIT_01_STA_4".M_CODES_UNIT_01_STA_4.M725) AND NOT "DB353_M_UNIT_01_STA_4".M_CODES_UNIT_01_STA_4.Ack_M725 AND NOT "DB2120_MPP_ITC_IPC".RESET_FAULTS AND NOT "DB353_M_UNIT_01_STA_4".M_CODES_UNIT_01_STA_4.M_RESET_PULSE;
END_REGION

REGION Network 29: READ-IN DISABLE / Read-in disable
   RUNG wire#powerrail
      Contact( "M_ONE" )
      wire#w1
      I_Contact( "DB353_M_UNIT_01_STA_4".M_CODES_UNIT_01_STA_4.M700 )
      I_Contact( "DB353_M_UNIT_01_STA_4".M_CODES_UNIT_01_STA_4.M702 )
      Not()
      Coil( "DB353_M_UNIT_01_STA_4".M_CODES_UNIT_01_STA_4.READ_IN_DISABLE_2 )
   END_RUNG
   RUNG wire#w1
      I_Contact( "DB353_M_UNIT_01_STA_4".M_CODES_UNIT_01_STA_4.READ_IN_DISABLE_2 )
      I_Contact( "DB353_M_UNIT_01_STA_4".M_CODES_UNIT_01_STA_4.M720 )
      I_Contact( "DB353_M_UNIT_01_STA_4".M_CODES_UNIT_01_STA_4.M722 )
      I_Contact( "DB353_M_UNIT_01_STA_4".M_CODES_UNIT_01_STA_4.M724 )
      I_Contact( "DB353_M_UNIT_01_STA_4".M_CODES_UNIT_01_STA_4.M725 )
      Not()
      Coil( "DB353_M_UNIT_01_STA_4".M_CODES_UNIT_01_STA_4.READ_IN_DISABLE_2 )
   END_RUNG
   RUNG wire#w1
      I_Contact( "DB353_M_UNIT_01_STA_4".M_CODES_UNIT_01_STA_4.READ_IN_DISABLE_2 )
      Not()
      Coil( "DB353_M_UNIT_01_STA_4".M_CODES_UNIT_01_STA_4.READ_IN_DISABLE_2 )
   END_RUNG
   RUNG wire#w1
      I_Contact( "DB353_M_UNIT_01_STA_4".M_CODES_UNIT_01_STA_4.READ_IN_DISABLE_2 )
      Not()
      Coil( "DB353_M_UNIT_01_STA_4".M_CODES_UNIT_01_STA_4.READ_IN_DISABLE_2 )
   END_RUNG
   // the same network as SCL:
   "DB353_M_UNIT_01_STA_4".M_CODES_UNIT_01_STA_4.READ_IN_DISABLE_2 := NOT ("M_ONE" AND NOT "DB353_M_UNIT_01_STA_4".M_CODES_UNIT_01_STA_4.M700 AND NOT "DB353_M_UNIT_01_STA_4".M_CODES_UNIT_01_STA_4.M702);
   "DB353_M_UNIT_01_STA_4".M_CODES_UNIT_01_STA_4.READ_IN_DISABLE_2 := NOT ("M_ONE" AND NOT "DB353_M_UNIT_01_STA_4".M_CODES_UNIT_01_STA_4.READ_IN_DISABLE_2 AND NOT "DB353_M_UNIT_01_STA_4".M_CODES_UNIT_01_STA_4.M720 AND NOT "DB353_M_UNIT_01_STA_4".M_CODES_UNIT_01_STA_4.M722 AND NOT "DB353_M_UNIT_01_STA_4".M_CODES_UNIT_01_STA_4.M724 AND NOT "DB353_M_UNIT_01_STA_4".M_CODES_UNIT_01_STA_4.M725);
   "DB353_M_UNIT_01_STA_4".M_CODES_UNIT_01_STA_4.READ_IN_DISABLE_2 := NOT ("M_ONE" AND NOT "DB353_M_UNIT_01_STA_4".M_CODES_UNIT_01_STA_4.READ_IN_DISABLE_2);
   "DB353_M_UNIT_01_STA_4".M_CODES_UNIT_01_STA_4.READ_IN_DISABLE_2 := NOT ("M_ONE" AND NOT "DB353_M_UNIT_01_STA_4".M_CODES_UNIT_01_STA_4.READ_IN_DISABLE_2);
END_REGION

REGION Network 30: READ-IN DISABLE / Read-in disable
   RUNG wire#powerrail
      Contact( "M_ONE" )
      wire#w1
      I_Contact( "DB353_M_UNIT_01_STA_4".M_CODES_UNIT_01_STA_4.READ_IN_DISABLE_2 )
      Not()
      Coil( "DB353_M_UNIT_01_STA_4".M_CODES_UNIT_01_STA_4.READ_IN_DISABLE_2 )
   END_RUNG
   RUNG wire#w1
      I_Contact( "DB353_M_UNIT_01_STA_4".M_CODES_UNIT_01_STA_4.READ_IN_DISABLE_2 )
      Not()
      Coil( "DB353_M_UNIT_01_STA_4".M_CODES_UNIT_01_STA_4.READ_IN_DISABLE_2 )
   END_RUNG
   RUNG wire#w1
      I_Contact( "DB353_M_UNIT_01_STA_4".M_CODES_UNIT_01_STA_4.READ_IN_DISABLE_2 )
      Not()
      Coil( "DB353_M_UNIT_01_STA_4".M_CODES_UNIT_01_STA_4.READ_IN_DISABLE_2 )
   END_RUNG
   RUNG wire#w1
      I_Contact( "DB353_M_UNIT_01_STA_4".M_CODES_UNIT_01_STA_4.READ_IN_DISABLE_2 )
      Not()
      Coil( "DB353_M_UNIT_01_STA_4".M_CODES_UNIT_01_STA_4.READ_IN_DISABLE_2 )
   END_RUNG
   // the same network as SCL:
   "DB353_M_UNIT_01_STA_4".M_CODES_UNIT_01_STA_4.READ_IN_DISABLE_2 := NOT ("M_ONE" AND NOT "DB353_M_UNIT_01_STA_4".M_CODES_UNIT_01_STA_4.READ_IN_DISABLE_2);
   "DB353_M_UNIT_01_STA_4".M_CODES_UNIT_01_STA_4.READ_IN_DISABLE_2 := NOT ("M_ONE" AND NOT "DB353_M_UNIT_01_STA_4".M_CODES_UNIT_01_STA_4.READ_IN_DISABLE_2);
   "DB353_M_UNIT_01_STA_4".M_CODES_UNIT_01_STA_4.READ_IN_DISABLE_2 := NOT ("M_ONE" AND NOT "DB353_M_UNIT_01_STA_4".M_CODES_UNIT_01_STA_4.READ_IN_DISABLE_2);
   "DB353_M_UNIT_01_STA_4".M_CODES_UNIT_01_STA_4.READ_IN_DISABLE_2 := NOT ("M_ONE" AND NOT "DB353_M_UNIT_01_STA_4".M_CODES_UNIT_01_STA_4.READ_IN_DISABLE_2);
END_REGION
END_FUNCTION
